{attribute 'TcGenerated'}
{attribute 'no-analysis'}
{attribute 'linkalways'}
// This function has been automatically generated from the project information.
VAR_GLOBAL CONSTANT
	{attribute 'const_non_replaced'}
	stLibVersion_STOBER_G6_Util : ST_LibVersion := (iMajor := 3, iMinor := 1, iBuild := 1, iRevision := 0, nFlags := 0, sVersion := '3.1.1.0');
END_VAR

(* stored: Version 1.1.0.1, ProductVersion 3.1.4024.6
   GVL Global_Version: Id {60fc244c-2bca-4801-9048-6a60eceee9ec} *)
